{attribute 'linkalways'} 
{attribute 'no_explicit_call' := 'This FB is a CLASS and must be accessed using methods or properties'}
{attribute 'enable_dynamic_creation'}
FUNCTION_BLOCK Node_F_VN_MedianElementElementwise_DINT EXTENDS VisionNode
VAR
    ipContainer : _ITcVnContainer;
    nMedian : _DINT(0);
    hrPrev : _HRESULT(S_OK);
    hresult : _HRESULT(S_OK);
END_VAR

METHOD PUBLIC  Clone : I_Node
VAR
	pNode : POINTER TO Node_F_VN_MedianElementElementwise_DINT;
END_VAR
pNode := __NEW(Node_F_VN_MedianElementElementwise_DINT);
Clone := pNode^;
END_METHOD

METHOD FB_init : BOOL
VAR_INPUT
	bInitRetains : BOOL; // if TRUE, the retain variables are initialized (warm start / cold start)
	bInCopyCode : BOOL;  // if TRUE, the instance afterwards gets moved into the copy code (online change)
END_VAR
AddInput('ipContainer', ipContainer);
AddInput('hrPrev', hrPrev);
AddOutput('ipContainer', ipContainer);
AddOutput('nMedian', nMedian);
AddOutput('hresult',hresult);
END_METHOD

METHOD PROTECTED OnExecute
hresult.Value := F_VN_MedianElementElementwise_DINT(
    ipContainer := ipContainer.Value,
    nMedian := nMedian.Value,
    hrPrev:= hrPrev.Value);
END_METHOD

METHOD PUBLIC PreExecutionCheck
VAR_INPUT
	Check : I_PreExecutionChecks;
END_VAR
Check.IsTrue(ipContainer.IsValid, 'ipContainer must be a valid container');
Check.IsTrue(ipContainer.IsType(TC_GLOBAL_CONST_LIST.ContainerType_Vector_DINT), 'ipContainer contains incorrect type');
END_METHOD

END_FUNCTION_BLOCK

(* stored: Version 1.1.0.1, ProductVersion 3.1.4026.18
   POU Node_F_VN_MedianElementElementwise_DINT: Id {5d81249a-d681-4370-80bd-d2e38c34a9ea}, SpecialFunc None
   Folder Constructor: Id {4399173c-f430-415b-bcd6-631a13819e8f}
   Method Clone: Id {933b2adc-4c7b-4256-9f1f-789ccec909fd}
   Method FB_init: Id {5bbe7ed8-9b01-4b17-9738-35639e1cf687}
   Method OnExecute: Id {4a5fee3e-99b5-404d-b80e-3f78cb5253bd}
   Method PreExecutionCheck: Id {1e63dd7b-a844-4a37-bf6f-878ff4f052dd} *)
